(* PLC project cmd_on_off_valve, Dassault Systèmes ControlBuild 2024x *)
(* stored: creationDateTime 2023-10-03T11:13:37-01:00 *)

FUNCTION_BLOCK actuator
  VAR_INPUT
    autoMode : BOOL := false;
    manualMode : BOOL := false;
  END_VAR
  VAR_INPUT
    autoCloseCmd : BOOL := false;
    autoOpenCmd : BOOL := false;
  END_VAR
  VAR_INPUT
    closedSensorFB : BOOL := false;
    openedSensorFB : BOOL := false;
  END_VAR
  VAR_INPUT
    closeValvePB : BOOL := false;
    openValvePB : BOOL := false;
  END_VAR
  VAR_INPUT
    generalFault : BOOL := false;
  END_VAR
  VAR_OUTPUT
    closeCmd : BOOL := false;
    openCmd : BOOL := false;
  END_VAR

(* LD diagram, written out as Structured Text *)
1:
openCmd := (autoMode AND autoOpenCmd AND NOT autoCloseCmd OR manualMode AND openValvePB AND NOT closeValvePB) AND NOT openedSensorFB AND NOT generalFault;
2:
closeCmd := (autoMode AND autoCloseCmd AND NOT autoOpenCmd OR manualMode AND closeValvePB AND NOT openValvePB) AND NOT closedSensorFB AND NOT generalFault;
END_FUNCTION_BLOCK

FUNCTION_BLOCK faults
  VAR_INPUT
    closeCmd : BOOL := false;
    openCmd : BOOL := false;
  END_VAR
  VAR_INPUT
    closedSensorFB : BOOL := false;
    openedSensorFB : BOOL := false;
  END_VAR
  VAR_INPUT
    acknowledgePB : BOOL := false;
  END_VAR
  VAR_OUTPUT
    generalFault : BOOL := false;
  END_VAR
  VAR
    closedSensorFault : BOOL := false;
    openedSensorFault : BOOL := false;
    discordanceFault : BOOL := false;
  END_VAR
  VAR
    ton_sec_1_i_ton : DINT := 0;
    ton_sec_1_t1_ton : REAL := 0.0;
    ton_sec_1_t2_ton : DINT := 0;
    ton_sec_1_Q : BOOL := false;
    ton_sec_1_CV : DINT := 0;
    ton_sec_2_i_ton : DINT := 0;
    ton_sec_2_t1_ton : REAL := 0.0;
    ton_sec_2_t2_ton : DINT := 0;
    ton_sec_2_Q : BOOL := false;
    ton_sec_2_CV : DINT := 0;
    ton_ms_3_i_tonms : DINT := 0;
    ton_ms_3_t1_tonms : REAL := 0.0;
    ton_ms_3_t2_tonms : DINT := 0;
    ton_ms_3_Q : BOOL := false;
    ton_ms_3_CV : DINT := 0;
  END_VAR
  VAR CONSTANT
    presetMvt : TIME := T#0h0m4s0ms;
    presetDiscordance : TIME := T#0h0m0s200ms;
  END_VAR

(* LD diagram, written out as Structured Text *)
1:
IF acknowledgePB THEN closedSensorFault := FALSE; END_IF;
IF acknowledgePB THEN openedSensorFault := FALSE; END_IF;
IF acknowledgePB THEN discordanceFault := FALSE; END_IF;
IF acknowledgePB THEN generalFault := FALSE; END_IF;
2:
TON_O(IN := openCmd, PT := presetMvt);
IF TON_O.Q0 AND NOT openedSensorFB THEN openedSensorFault := TRUE; END_IF;
TON_C(IN := closeCmd, PT := presetMvt);
IF TON_C.Q0 AND NOT closedSensorFB THEN closedSensorFault := TRUE; END_IF;
3:
TON_DISC(IN := openedSensorFB AND closedSensorFB, PT := presetDiscordance);
IF TON_DISC.Q0 THEN discordanceFault := TRUE; END_IF;
4:
IF closedSensorFault OR openedSensorFault OR discordanceFault THEN generalFault := TRUE; END_IF;
END_FUNCTION_BLOCK

(* Command of an on/off valve with fault detection. *)
PROGRAM cmd_equipment_library.cmd_on_off_valve
  VAR_INPUT
    autoMode : BOOL := false;
    manualMode : BOOL := false;
  END_VAR
  VAR_INPUT
    closedSensorFB : BOOL := false;
    openedSensorFB : BOOL := false;
  END_VAR
  VAR_INPUT
    autoCloseCmd : BOOL := false;
    autoOpenCmd : BOOL := false;
  END_VAR
  VAR_INPUT
    closeValvePB : BOOL := false;
    openValvePB : BOOL := false;
  END_VAR
  VAR_INPUT
    acknowledgePB : BOOL := false;
  END_VAR
  VAR_OUTPUT
    closeCmd : BOOL := false;
    openCmd : BOOL := false;
  END_VAR
  VAR_OUTPUT
    generalFault : BOOL := false;
  END_VAR

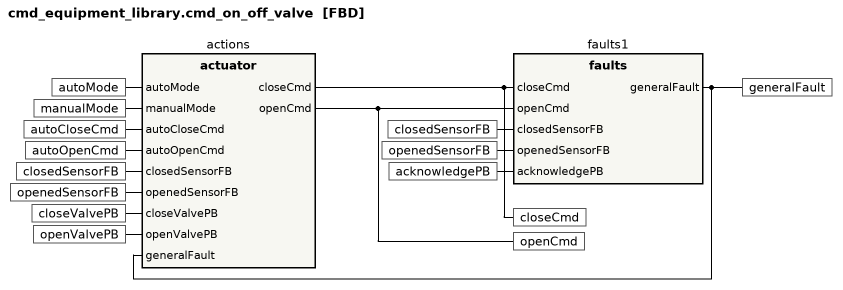
(* FBD diagram, written out as Structured Text *)
faults1(closeCmd := actions.closeCmd, openCmd := actions.openCmd, closedSensorFB := closedSensorFB, openedSensorFB := openedSensorFB, acknowledgePB := acknowledgePB);
actions(autoMode := autoMode, manualMode := manualMode, autoCloseCmd := autoCloseCmd, autoOpenCmd := autoOpenCmd, closedSensorFB := closedSensorFB, openedSensorFB := openedSensorFB, closeValvePB := closeValvePB, openValvePB := openValvePB, generalFault := faults1.generalFault);
closeCmd := actions.closeCmd;
openCmd := actions.openCmd;
generalFault := faults1.generalFault;
END_PROGRAM
